PROGRAM ReadAnalogInput
VAR
	Temp: REAL;
END_VAR

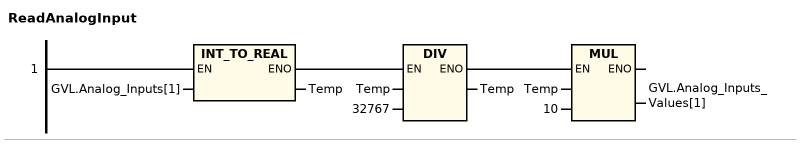
// NETWORK 1
Temp := INT_TO_REAL(GVL.Analog_Inputs[1]);
Temp := Temp / 32767;
GVL.Analog_Inputs_Values[1] := Temp * 10;

END_PROGRAM

(* stored: Version 1.1.0.1, ProductVersion 3.1.4024.12
   POU ReadAnalogInput: Id {00ecc9df-f4bc-4d10-b751-3d1ddc05503e}, SpecialFunc None *)
